// TIA Portal V17 export
// export: Created 2021-12-03T08:13:15.1987524Z, ExportSetting WithDefaults, DisplayName Totally Integrated Automation Portal, DisplayVersion V17, DisplayName TIA Portal Openness, DisplayVersion V17, DisplayName TIA Portal Version Control Interface, DisplayVersion V17, DisplayName STEP 7 Professional, DisplayVersion V17, DisplayName STEP 7 Safety, DisplayVersion V17, DisplayName WinCC Advanced, DisplayVersion V17
DATA_BLOCK "FGDB_Outputs"   // DB60, F_DB
VERSION : 0.1
// stored: AutoNumber false
   VAR
      O_PowerModulator : Bool;   // 400 VAC Power Modulator NA2-1Q3
      O_PowerChiller : Bool;   // 400 VAC Power Chiller NA2-1Q5
      O_PowerConveyor : Bool;   // 400 VAC Power Conveyor NA2-1Q7
      O_PowerXRayUnit : Bool;   // 230 VAC Power X-Ray Unit NA2-2Q7
      O_PowerModulator1P : Bool;   // 230 VAC Power Modulator
      O_ChilVlv_PwrOn : Bool;   // 230 VAC Power Chiller Valve
      O_ModSwic_PwrOn : Bool;   // 230 VAC Power Modulator Switch
      O_AccIntrlck : Bool;   // Interlock Accelerator
      O_SpareIntrlck : Bool;   // Interlock Spare
   END_VAR
BEGIN
END_DATA_BLOCK
